// TIA Portal V20 export
TYPE "LER_typeSleep"
// stored: Access Published
   STRUCT
      Servo : Struct
         sleep : Bool;
         deppSleep : Bool;
      END_STRUCT;
      MotionPower : Struct
         sleep : Bool;
         deppSleep : Bool;
      END_STRUCT;
      FFU : Struct
         sleep : Bool;
         deppSleep : Bool;
         data : Int;
      END_STRUCT;
      RingBlower : Struct
         sleep : Bool;
         deppSleep : Bool;
         data : Real;
      END_STRUCT;
      Heater : Struct
         sleep : Bool;
         deppSleep : Bool;
         data : Int;
      END_STRUCT;
   END_STRUCT;
END_TYPE
